FUNCTION_BLOCK IED64 (* Earth Fault Protection device *)
  (* Standard: 61499-2; ApplicationDomain: Smart Grid Protection Systems; Function: Earth Fault Protection IED; Type: IED; Description: Earth Fault protection Intelligent Electronic Device (IED) type 64. *)
  (* Version 1.0, 24.02.2021, badger, AUT, Redesign of the earth fault IED from Gulnara's original design. *)
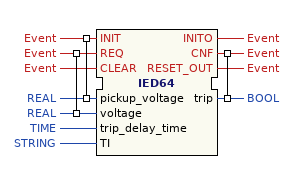
  EVENT_INPUT
    INIT WITH pickup_voltage; (* Initialization Request *)
    REQ WITH voltage; (* Reads the voltage from the substation *)
    CLEAR; (* External signal to manually clear a tripped IED *)
  END_EVENT
  EVENT_OUTPUT
    INITO; (* Initialization Confirm *)
    CNF WITH trip; (* Execution Confirmation *)
    RESET_OUT; (* Signals that the IED has been reset after the earth fault has been cleared *)
  END_EVENT
  VAR_INPUT
    pickup_voltage : REAL := 0; (* The voltage from the earth fault that defines the trip point for the IED *)
    voltage : REAL := 0; (* Earth leakage voltage from the substation interface *)
    trip_delay_time : TIME; (* Time in milliseconds after a fault before the IED is tripped. *)
    TI : STRING; (* Requirements Traceability ID *)
  END_VAR
  VAR_OUTPUT
    trip : BOOL := false; (* True if the IED has been tripped by an earth fault *)
  END_VAR
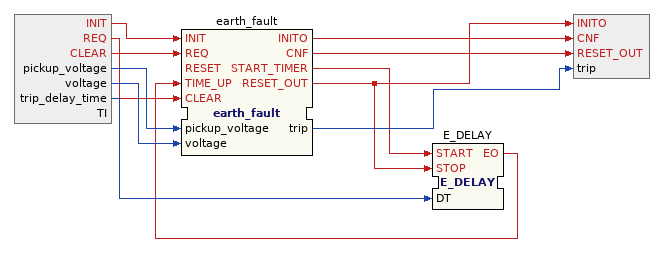
  FBS
    E_DELAY : E_DELAY;
    earth_fault : earth_fault;
  END_FBS
  EVENT_CONNECTIONS
    INIT TO earth_fault.INIT;
    REQ TO earth_fault.REQ;
    E_DELAY.EO TO earth_fault.TIME_UP;
    CLEAR TO earth_fault.CLEAR;
    earth_fault.INITO TO INITO;
    earth_fault.CNF TO CNF;
    earth_fault.START_TIMER TO E_DELAY.START;
    earth_fault.RESET_OUT TO E_DELAY.STOP;
    earth_fault.RESET_OUT TO RESET_OUT;
  END_CONNECTIONS
  DATA_CONNECTIONS
    trip_delay_time TO E_DELAY.DT;
    pickup_voltage TO earth_fault.pickup_voltage;
    voltage TO earth_fault.voltage;
    earth_fault.trip TO trip;
  END_CONNECTIONS
END_FUNCTION_BLOCK
